(* CODESYS project http.20210810.1.project

Project tree, tasks and I/O mapping:
  MIC7001 : Changsha-Cyber-MI-linux, Changsha Cyber-MI Co., Ltd., version 3.5.10.40
    application Application
      libraries: Standard, * (System); CAA Types Extern, * (CAA Technical Workgroup); CAA Callback Extern, * (CAA Technical Workgroup); SysMem, * (System); SysTypes Interfaces, * (System); SysTime, * (System); CAA DTUtil Extern, 3.5.12.0 (CAA Technical Workgroup); CAA Real Time Clock Extern, 3.5.10.0 (CAA Technical Workgroup); CAN API, 1.0.0.3 (3S - Smart Software Solutions GmbH); SysFile, 3.5.15.0 (System); AC_DataLog, 3.5.14.0 (3S - Smart Software Solutions GmbH); CAA Net Base Services, 3.5.15.0 (CAA Technical Workgroup); CAA Memory, 3.5.12.0 (CAA Technical Workgroup); CAA SerialCom, 3.5.15.0 (CAA Technical Workgroup); Util, 3.5.15.0 (System); CAA Can Low Level Imp Extern, 3.5.11.0 (CAA Technical Workgroup); CAA Can Low Level Extern, 3.5.15.0 (CAA Technical Workgroup); VisuDialogs, * (System); CmpBitmapPool, * (System); CAA File, 3.5.15.0 (CAA Technical Workgroup); IODrvEtherCAT, 3.5.15.50 (3S - Smart Software Solutions GmbH); SysShm Implementation, 3.5.16.0 (System); SysShm, 3.5.8.0 (System); MIC7001 base library, 1.11 (Cyber-MI.com); HTTP Client, 1.0.1.2 (CODESYS GmbH)
      task VISU_TASK (cyclic, interval 100 ms, priority 31) calls nothing
      program prg_http_client [ST]
    SoftMotion General Axis Pool
  libraries: CmpBitmapPool, * (System)
  5ce3da45-db07-42e7-a21c-a00fff4ed8f6|D:\工作文件\009中集集团\DOCS\等油耗图.jpg
  5ce3da45-db07-42e7-a21c-a00fff4ed8f6|C:\Users\RJST\Desktop\bmp1.png
  text list GlobalTextList
*)

// MIC7001/Application/prg_http_client
PROGRAM prg_http_client
VAR
	http_client:HTTP.httpclient();
END_VAR



http_client();

END_PROGRAM
